(* IEC 61131-3 sources: plc_generation_empirical_study/datasets/packages/internal_v0_1/qualification_only/C09_E01_latched_alarm_acknowledge, 1 file *)

(* ---- reference.st ---- *)
FUNCTION_BLOCK C09_E01_latched_alarm_acknowledge
VAR_INPUT
    AlarmCondition : BOOL;
    Acknowledge : BOOL;
    Reset : BOOL;
END_VAR
VAR_OUTPUT
    AlarmActive : BOOL;
    AlarmUnacked : BOOL;
END_VAR

IF AlarmCondition THEN
    AlarmActive := TRUE;
    AlarmUnacked := TRUE;
ELSE
    IF Acknowledge THEN
        AlarmUnacked := FALSE;
    END_IF;
    IF Reset THEN
        AlarmActive := FALSE;
        AlarmUnacked := FALSE;
    END_IF;
END_IF;

END_FUNCTION_BLOCK
